TYPE ST_System_BWK_Steuerung :
STRUCT
	Freigabe				: ST_Steuerung_auto_manu_BOOL;
	Freigabe_Deakt		: ST_Steuerung_auto_manu_BOOL;
	Betrieb_Anford		: ST_Steuerung_auto_manu_opti_BOOL;

	Regelung_Sollw		: ST_Steuerung_auto_manu_opti_REAL;

	Quittierung			: BOOL;
END_STRUCT
END_TYPE

(* stored: Version 1.1.0.1, ProductVersion 3.1.4024.9
   DUT ST_System_BWK_Steuerung: Id {1b15bbd4-2364-415b-9db0-d55547f0c5e2} *)
